PROGRAM MAIN
VAR
	bInit			: 	BOOL	:=FALSE;
	bStatus			:	BOOL;
	PosControl		:	MotionControl;
	
END_VAR

IF NOT bInit THEN
	

	bInit	:=TRUE;
END_IF

END_PROGRAM

(* stored: Version 1.1.0.1, ProductVersion 3.1.4024.11
   POU MAIN: Id {4d21455b-79d8-4b20-82b7-7fb4a300dc2a}, SpecialFunc None *)
